PROGRAM P_CameraFlip
VAR
	fbFileOpen: FB_FileOpen;
    fbFileWrite: FB_FileWrite;
    fbFileClose: FB_FileClose;
    hFile : UINT;
    nResultCreate, nResultDelete : INT;
    sPath : STRING := 'C:\Users\Administrator\Desktop\CameraFlip\trigger.txt';
    bFileExists : BOOL;
	Step:INT;
	ftrig:F_trig;
	RisingEdge:R_trig;
	bBusy 				:BOOL;
	bError				:BOOL;
	nErrId				:UDINT;
    nIndex				:INT;
END_VAR

RisingEdge(CLK := gvl_error.b_cameras_ivms);

CASE Step OF
    0:
        // Jeśli wystąpiło zdarzenie zapisu lub zmiany receptury
        IF RisingEdge.Q THEN
            bBusy := TRUE;
            bError := FALSE;
            nErrId := 0;
            nIndex := 0;

            Step := 10;  
        END_IF

    10:

            fbFileOpen(
                sNetId := '', 
                sPathName := sPath, 
                nMode := FOPEN_MODEAPPEND OR FOPEN_MODETEXT, 
                ePath := PATH_GENERIC, 
                bExecute := TRUE
            );      
        Step := 20;

    20:
        // Czekaj na otwarcie pliku
        fbFileOpen(bExecute := FALSE);
        IF NOT fbFileOpen.bBusy THEN
            IF fbFileOpen.bError THEN
                nErrId := fbFileOpen.nErrId;
                bError := TRUE;
                Step := 500;  
            ELSE
                hFile := fbFileOpen.hFile;
                Step := 300;  
            END_IF
        END_IF 

    300:
        // Zamknij plik
        fbFileClose(
            sNetId := '', 
            hFile := hFile, 
            bExecute := TRUE
        );
        Step := 310;

    310:
        // Czekaj na zamknięcie pliku
        fbFileClose(bExecute := FALSE);
        IF NOT fbFileClose.bBusy THEN
            IF fbFileClose.bError THEN
                nErrId := fbFileClose.nErrId;
                bError := TRUE;
            END_IF
            Step := 500;  
        END_IF

    500:
        bBusy := FALSE;
        Step := 0;
END_CASE

END_PROGRAM

(* stored: Version 1.2.0.0, ProductVersion 3.1.4026.13, FileIdentifier f27ba1a65a6198171f7783fae94443682b736b62, FileSignature 89611f707a0b902c5c9c5e92b83696e8df6b382ab498a3e0a47882bccff6fa16f005d418476e59f4bf7025f128e8e280255a789ced9527f2bd7f7bb54520f34f60f31ae6a96ce18d51372b4115d986f5146b12f0ccf6a2e95827e1b036ff1bf6d97f2eb3d771d1d28b52e4bec3a88561e959d8d161f3556d6518a8e9b6d641162327a72677aeeb6b9b60a1af81e272b75d4305a1383c316ba3eb9ba1aa71e73b9076ad6633cf7f02d178d5fcb46c88383a37a258ab4293115d04cecebb777cc3e6da11c24d20adc7cea8f7365c1d0e58036974eefc64fd8d97acf3de7e0cbdfc836cf815cbfbc48cb6c0d845246cc3fdd439b6a4ffa5b8f95ade4f49d1b5f508
   POU P_CameraFlip: Id {d37b2de1-8934-4578-8b9b-edb828947d13}, SpecialFunc None *)
